// TwinCAT 3 PLC project CommunicatorApp
// ProgramVersion: 3.1.4023.0
// libraries:
//   Tc2_Standard, * (Beckhoff Automation GmbH)
//   Tc2_System, * (Beckhoff Automation GmbH)
//   Tc2_Utilities, * (Beckhoff Automation GmbH)
//   Tc3_IotCommunicator, * (Beckhoff Automation GmbH)
//   Tc3_Module, * (Beckhoff Automation GmbH)
// project tree:
//   DUTs/ ST_DataRoom1.TcDUT, ST_DataRoom2.TcDUT
//   / PlcTask.TcTTO
//   POUs/ MAIN.TcPOU, P_FreeRoom.TcPOU, P_FreeRoom2.TcPOU
// real-time tasks:
//   TASK PlcTask: cycle T#10ms, priority 20, ADS port 350

CONFIGURATION CommunicatorApp
    RESOURCE PLC ON TwinCAT3
        TASK PlcTask(INTERVAL := T#10ms, PRIORITY := 20);
        PROGRAM MAIN WITH PlcTask : MAIN;
    END_RESOURCE
END_CONFIGURATION

// ---- DUTs/ST_DataRoom1.TcDUT
TYPE ST_DataRoom1 :
STRUCT
    {attribute 'iot.DisplayName' := 'Temperature 1'}
    {attribute 'iot.ReadOnly' := 'true'}
    {attribute 'iot.Unit' := 'Celsius'}
    {attribute 'iot.MinValue' := '5'}
    {attribute 'iot.MaxValue' := '30'}
    nTemp1  : REAL;
    {attribute 'iot.DisplayName' := 'Temperature 2'}
    {attribute 'iot.ReadOnly' := 'true'}
    {attribute 'iot.Unit' := 'Celsius'}
    {attribute 'iot.MinValue' := '5'}
    {attribute 'iot.MaxValue' := '30'}
    nTemp2  : REAL;
    {attribute 'iot.DisplayName' := 'Temperature 3'}
    {attribute 'iot.ReadOnly' := 'true'}
    {attribute 'iot.Unit' := 'Celsius'}
    {attribute 'iot.MinValue' := '5'}
    {attribute 'iot.MaxValue' := '30'}
    nTemp3  : REAL;
	{attribute 'iot.DisplayName' := 'Some value with range'}
    //{attribute 'iot.ReadOnly' := 'true'}
    {attribute 'iot.Unit' := 'some unit'}
    {attribute 'iot.MinValue' := '-20'}
    {attribute 'iot.MaxValue' := '70'}
    nSetValue  : REAL;
	
END_STRUCT
END_TYPE

// ---- DUTs/ST_DataRoom2.TcDUT
TYPE ST_DataRoom2 :
STRUCT
	
	{attribute 'iot.DisplayName' := 'Start/Stop Blinker'}
    bBlinker1 : BOOL;
    {attribute 'iot.DisplayName' := 'Im blinking'}
	{attribute 'iot.ReadOnly' := 'true'}
    bBlinker2 : BOOL;
	
	{attribute 'iot.DisplayName' := 'Start/Stop Counting'}
    bCount : BOOL;
    {attribute 'iot.DisplayName' := 'Counting'}
	{attribute 'iot.ReadOnly' := 'true'}
    bCount2 : BOOL;
	
    {attribute 'iot.DisplayName' := 'Going Up'}
	{attribute 'iot.ReadOnly' := 'true'}
	{attribute 'iot.Unit' := 'integer'}	
	uiSomeValue : UINT;
	
    {attribute 'iot.DisplayName' := 'Going Up 2'}
	{attribute 'iot.ReadOnly' := 'true'}
	{attribute 'iot.Unit' := 'real'}	
	rSomeValue : REAL;
	
	{attribute 'iot.DisplayName' := 'Reset'}
    bReset : BOOL;
	
	
END_STRUCT
END_TYPE

// ---- POUs/MAIN.TcPOU
PROGRAM MAIN
VAR
END_VAR

P_FreeRoom();
P_FreeRoom2();

END_PROGRAM

// ---- POUs/P_FreeRoom.TcPOU
// Beckhoff Polska
// przykladowy program do obslugi TF6730 IoT_Communicator
// Wymaga dodania bibliotek Tc3_IoTCommunicator oraz Tc2_Utilities
// v1.0
// 22/08/2019
PROGRAM P_FreeRoom
VAR
	fbIoT			: FB_IotCommunicator := (
						sHostName	:= '127.0.0.1',
						nPort		:= 1883,
						sMainTopic	:= 'MyMainTopic',
						sDeviceName	:= 'Room One');
	stData			: ST_DataRoom1;
	timer			: TON;
	fbRand			: DRAND;
	fbGetTime		: NT_GetTime;
	bSendMessage	: BOOL;
	sMessage		: STRING(255) := 'my plc message';
	wSeed			: WORD;
	nDummy: REAL;
END_VAR


// keep alive
fbIoT.Execute(TRUE);

timer(IN := NOT timer.Q, PT := T#500MS);


// synchronize data
IF fbIoT.bConnected AND timer.Q THEN
    fbIoT.SendData(ADR(stData), SIZEOF(stData));
END_IF


// pending changes from Android App
IF fbIoT.fbCommand.bAvailable THEN
    IF fbIoT.fbCommand.sVarName = 'nSetValue' THEN
		fbIoT.fbCommand.GetValue(ADR(stData.nSetValue), SIZEOF(stData.nSetValue), E_IotCommunicatorDatatype.type_REAL);
		IF (stData.nSetValue > 70 ) THEN
			stData.nSetValue := 70;
			fbIoT.SendMessage('Set temperature too high!!! Max temp is 70.');
		ELSIF (stData.nSetValue < -20 ) THEN	
			stData.nSetValue := -20;
			fbIoT.SendMessage('Set temperature too low!!! Min temp is -20.');
		END_IF
    END_IF
    fbIoT.fbCommand.Remove();
END_IF


// rand temp
fbGetTime(START := timer.Q);
wSeed := fbGetTime.TIMESTR.wMinute + fbGetTime.TIMESTR.wSecond + fbGetTime.TIMESTR.wMilliseconds;

IF timer.Q THEN
	// temp1
	fbRand(Seed := WORD_TO_INT(wSeed));
	stData.nTemp1 := stData.nTemp1 + (fbRand.Num - 0.5);
	stData.nTemp1 := INT_TO_REAL(REAL_TO_INT(stData.nTemp1 * 100))/100; // cut off last digits
	IF (stData.nTemp1 < 5) THEN
		stData.nTemp1 := 5;
	ELSIF (stData.nTemp1 > 30) THEN
		stData.nTemp1 := 30;
	END_IF
	// temp2
	fbRand(Seed := WORD_TO_INT(wSeed + 1));
	stData.nTemp2 := stData.nTemp2 + (fbRand.Num - 0.5);
	stData.nTemp2 := INT_TO_REAL(REAL_TO_INT(stData.nTemp2 * 100))/100; // cut off last digits
	IF (stData.nTemp2 < 5) THEN
		stData.nTemp2 := 5;
	ELSIF (stData.nTemp2 > 30) THEN
		stData.nTemp2 := 30;
	END_IF
	// temp 3
	fbRand(Seed := WORD_TO_INT(wSeed + 2));
	stData.nTemp3 := stData.nTemp3 + (fbRand.Num - 0.5);
	stData.nTemp3 := INT_TO_REAL(REAL_TO_INT(stData.nTemp3 * 100))/100; // cut off last digits
	IF (stData.nTemp3 < 5) THEN
		stData.nTemp3 := 5;
	ELSIF (stData.nTemp3 > 30) THEN
		stData.nTemp3 := 30;
	END_IF
END_IF


// send plc message
IF bSendMessage THEN
	bSendMessage := FALSE;
	fbIoT.SendMessage(sMessage);
END_IF


nDummy := stData.nSetValue - REAL_TO_INT(stData.nSetValue);

END_PROGRAM

// ---- POUs/P_FreeRoom2.TcPOU
// Beckhoff Polska
// przykladowy program do obslugi TF6730 IoT_Communicator
// Wymaga dodania bibliotek Tc3_IoTCommunicator oraz Tc2_Utilities
// v1.0
// 22/08/2019
PROGRAM P_FreeRoom2
VAR
	fbIoT 			: FB_IotCommunicator := (
						sHostName := '127.0.0.1',
						nPort := 1883,
						sMainTopic := 'MyMainTopic',
						sDeviceName := 'Room 2');
	stData			: ST_DataRoom2;
	timer			: TON;
	timer2			: TON;
	timer3			: TON;
	rTrig			: R_TRIG;
	fTrig			: F_TRIG;
	rTrigReset		: R_TRIG;
	fbRand			: DRAND;
	bSendMessage	: BOOL;
	sMessage		: STRING(255) := 'my plc message 2';

END_VAR


// keep alive
fbIoT.Execute(TRUE);

timer(	IN := NOT timer.Q, 	PT := T#500MS);
timer2(	IN := NOT timer2.Q, PT := T#2S);


// synchronize data
IF fbIoT.bConnected AND timer.Q THEN
    fbIoT.SendData(ADR(stData), SIZEOF(stData));
END_IF


// pending changes from Android App
IF fbIoT.fbCommand.bAvailable THEN
	IF fbIoT.fbCommand.sVarName = 'bBlinker1' THEN
		fbIoT.fbCommand.GetValue(	ADR(stData.bBlinker1),
									SIZEOF(stData.bBlinker1),
									E_IotCommunicatorDatatype.type_BOOL);
	ELSIF fbIoT.fbCommand.sVarName = 'bCount' THEN
		fbIoT.fbCommand.GetValue(	ADR(stData.bCount),
									SIZEOF(stData.bCount),
									E_IotCommunicatorDatatype.type_BOOL);
	ELSIF fbIoT.fbCommand.sVarName = 'bReset' THEN
		fbIoT.fbCommand.GetValue(	ADR(stData.bReset),
									SIZEOF(stData.bReset),
									E_IotCommunicatorDatatype.type_BOOL);
					
	END_IF
	fbIoT.fbCommand.Remove();
END_IF


// reset counter
IF stData.bReset THEN	
	stData.bReset := FALSE;
	stData.bCount := FALSE;
	stData.bCount2 := FALSE;
	stData.rSomeValue := 0;
	stData.uiSomeValue := 0;
	fbIoT.SendMessage('Reset Counter');
END_IF


// blink some bool
IF stData.bBlinker1 AND timer2.Q THEN
	stData.bBlinker2 := NOT stData.bBlinker2;
ELSIF NOT stData.bBlinker1 AND timer2.Q THEN
	stData.bBlinker2 := FALSE;
END_IF


//cont int and real
rTrig(CLK := stData.bCount);
IF rTrig.Q THEN
	stData.bCount2 := TRUE;
	fbIoT.SendMessage('Counting Started');	
END_IF
fTrig(CLK := stData.bCount);
IF fTrig.Q THEN
	stData.bCount2 := FALSE;
	fbIoT.SendMessage('Counting Stopped');
END_IF
IF stData.bCount2 THEN
	fbRand(Seed := UINT_TO_INT(stData.uiSomeValue));
	stData.rSomeValue := stData.rSomeValue + LREAL_TO_REAL(fbRand.Num);
	stData.uiSomeValue := stData.uiSomeValue + 1;
END_IF


// send plc message
IF bSendMessage THEN
	bSendMessage := FALSE;
	fbIoT.SendMessage(sMessage);
END_IF

END_PROGRAM
